FUNCTION_BLOCK FB_DeletePartProgram 
VAR_INPUT
	Execute 	: BOOL;
	sNetId		: STRING;
	sPathName	: STRING;
	filesList   : ARRAY[0..99] OF STRING;
	filesNumb	: UINT;
END_VAR
VAR_OUTPUT
	Busy : BOOL;
	Done : BOOL;
	Error : BOOL;
	ErrorID : DINT;
	ErrorSubID : UDINT;
END_VAR
VAR
	iState : DINT := -1;
	i : USINT;
	fbFileDelete: FB_FileDelete;
	RTRIG_Execute : R_TRIG;
	TON_Timeout		: TON;
END_VAR

TON_Timeout(IN := Busy, PT := T#20S);
IF TON_Timeout.Q THEN
	
	iState := 1999;
END_IF

RTRIG_Execute(CLK := Execute);
IF(RTRIG_Execute.Q) THEN
	Done := FALSE;
	i := 0;
	ErrorID := 0;
	ErrorSubID := 0;
	
	iState := 0;
ELSIF NOT Execute AND NOT Busy THEN
	Busy			:= FALSE;
	Done			:= FALSE;
	Error			:= FALSE;
	
	iState := -1;
END_IF

CASE iState OF
	-1:
		;
	0:
		Busy := TRUE;
		fbFileDelete.sPathName := CONCAT(sPathName,filesList[i]);
		iState := 10;
		
	10:
		fbFileDelete.bExecute := TRUE;
		iState := 20;
			
	20:
        fbFileDelete.bExecute := FALSE; 
        IF NOT fbFileDelete.bBusy THEN 
        	IF fbFileDelete.bError THEN 
            	ErrorSubID := fbFileDelete.nErrId; 
                iState := 1020;
               ELSE 
                 	iState := 30;
               END_IF 
          END_IF
		  
	30:
		i := i + 1;
		IF i < filesNumb AND i <= 99 THEN
			iState := 0;
		ELSE
			iState := 999;
		END_IF

	999:
		Busy	 			:= FALSE;
		Done				:= TRUE;
	
		iState := -1;	
END_CASE

IF(iState > 999) THEN
	Error 	:= TRUE;
	ErrorID := iState;
	Busy 	:= FALSE;
ELSE
	Error := FALSE;
END_IF

A_Call();

ACTION A_Call:
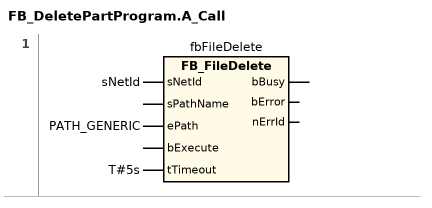
// NETWORK 1
fbFileDelete(sNetId := sNetId, ePath := PATH_GENERIC, tTimeout := T#5s); // FB_FileDelete
END_ACTION

END_FUNCTION_BLOCK

(* stored: Version 1.1.0.1, ProductVersion 3.1.4024.13
   POU FB_DeletePartProgram: Id {85ed054c-cb8a-4f09-a83a-a46cb0b7417c}, SpecialFunc None
   Action A_Call: Id {e1f42e70-5a41-4d5e-a93a-04ed5770413c} *)
